Yaskawa INFORM job: JOB0014.JBI

/JOB
//NAME JOB0014
//POS
///NPOS 32,32,0,0,0,0
///POSTYPE PULSE
///PULSE
///TOOL 0
C00000=0,-72817,-54613,0,7281,0
C00001=92160,-72817,-54613,0,7281,0
C00002=92160,-72817,-54613,0,21845,0
C00003=92353,-45256,-11058,125,13222,-85
C00004=92353,-45256,-11058,125,13222,-85
C00005=92353,-45256,-11058,125,13222,-85
C00006=92353,-45256,-11058,125,13222,-85
C00007=92353,-45256,-11058,125,13222,-85
C00008=92353,-39432,-439,199,8221,-126
C00009=92353,-41285,-3745,168,9755,-109
C00010=92372,-32954,-1382,91,12863,-61
C00011=92353,-45256,-11058,125,13222,-85
C00012=92353,-45256,-11058,125,13222,-85
C00013=92353,-45256,-11058,125,13222,-85
C00014=92353,-45256,-11058,125,13222,-85
C00015=92353,-45256,-11058,125,13222,-85
C00016=92353,-45256,-11058,125,13222,-85
C00017=92353,-39432,-439,199,8221,-126
C00018=92353,-41285,-3745,168,9755,-109
C00019=92372,-32954,-1382,91,12863,-61
C00020=92353,-45256,-11058,125,13222,-85
C00021=92353,-51940,-24538,84,19996,-61
C00022=92353,-45256,-11058,125,13222,-85
C00023=92353,-45256,-11058,125,13222,-85
C00024=92353,-45256,-11058,125,13222,-85
C00025=92353,-45256,-11058,125,13222,-85
C00026=92353,-45256,-11058,125,13222,-85
C00027=92353,-45256,-11058,125,13222,-85
C00028=92353,-45256,-11058,125,13222,-85
C00029=92160,-72817,-54613,0,21845,0
C00030=92160,-72817,-54613,0,7281,0
C00031=0,-72817,-54613,0,7281,0
BC00000=1675539,-209806,0
BC00001=1675539,-209806,0
BC00002=1675539,-209806,0
BC00003=1675539,-209806,0
BC00004=1675539,-209806,-1555432
BC00005=1675539,-209806,-1555432
BC00006=1675539,-209806,-1555432
BC00007=1675539,-209806,-1555432
BC00008=1675539,-209806,-1555432
BC00009=1675539,-209806,-1555432
BC00010=1675539,-209806,-1555432
BC00011=1675539,-209806,-1555432
BC00012=1675539,-209806,-1555432
BC00013=1965453,-211082,-1555432
BC00014=1965453,-211082,-1555432
BC00015=1965453,-211082,-1555432
BC00016=1965453,-211082,-1555432
BC00017=1965453,-211082,-1555432
BC00018=1965453,-211082,-1555432
BC00019=1965453,-211082,-1555432
BC00020=1965453,-211082,-1555432
BC00021=1965517,-196539,-1606631
BC00022=1965299,-246191,-1606631
BC00023=1965299,-246191,-1504232
BC00024=1965608,-175972,-1606631
BC00025=1675384,-244915,-1606631
BC00026=1675603,-195263,-1534224
BC00027=1675603,-195263,-1534224
BC00028=1675603,-195263,0
BC00029=1675603,-195263,0
BC00030=1675603,-195263,0
BC00031=1675603,-195263,0
//INST
///DATE 2026/01/17 21:54
///ATTR SC,RW
///GROUP1 RB1,BS1
NOP
'2026/01/17 21:54
CALL JOB:HOME
MOVJ C00000 BC00000 VJ=100.00
MOVJ C00001 BC00001 VJ=100.00
MOVJ C00002 BC00002 VJ=100.00
MOVJ C00003 BC00003 VJ=100.00
MOVL C00004 BC00004 V=500.0
'SEARCH S-END
MOVL C00005 BC00005 V=500.0
REFP 3 C00006 BC00006
REFP 4 C00007 BC00007
REFP 5 C00008 BC00008
REFP 6 C00009 BC00009
REFP 7 C00010 BC00010
CALL JOB:B-SRCH3
SET P021 P006
SFTOF
MOVL C00011 BC00011 V=500.0
SFTON P021
MOVL C00012 BC00012 V=500.0
MOVL C00013 BC00013 V=500.0
SFTOF
'SEARCH S-START
MOVL C00014 BC00014 V=500.0
REFP 3 C00015 BC00015
REFP 4 C00016 BC00016
REFP 5 C00017 BC00017
REFP 6 C00018 BC00018
REFP 7 C00019 BC00019
CALL JOB:B-SRCH3
SET P020 P006
SFTOF
MOVL C00020 BC00020 V=500.0
PULSE OT#(4096) T=0.5
'WELD Weld_0074
SFTON P020
MOVL C00021 BC00021 V=500.0
MOVL C00022 BC00022 V=200.0
ARCON ASF#(3)
REFP 1 C00023 BC00023
REFP 2 C00024 BC00024
COMARCON WEV#(3) U/D=320 L/R=0.0
SFTON P021
MOVL C00025 BC00025
COMARCOF
ARCOF
MOVL C00026 BC00026 V=200.0
SFTOF
MOVL C00027 BC00027 V=500.0
MOVL C00028 BC00028 V=500.0
MOVJ C00029 BC00029 VJ=100.00
MOVJ C00030 BC00030 VJ=100.00
MOVJ C00031 BC00031 VJ=100.00
CALL JOB:HOME
END
